FUNCTION_BLOCK Seven_State_Actuator_CAT (* Composite Function Block Type *)
  (* Standard: 61499-2 *)
  (* Version 0.0, 10/7/2025, Schneider Electric, template *)
  PACKAGE Main;
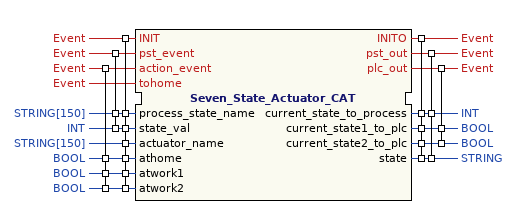
  EVENT_INPUT
    INIT WITH process_state_name, state_val, actuator_name, athome, atwork1, atwork2; (* Initialization Request *)
    pst_event WITH process_state_name, state_val;
    action_event WITH athome, atwork1, atwork2;
    tohome;
  END_EVENT
  EVENT_OUTPUT
    INITO WITH current_state_to_process, current_state1_to_plc, current_state2_to_plc, state; (* Initialization Confirm *)
    pst_out WITH current_state_to_process, state; (* Initialization Confirm *)
    plc_out WITH current_state1_to_plc, current_state2_to_plc;
  END_EVENT
  VAR_INPUT
    process_state_name : STRING[150];
    state_val : INT;
    actuator_name : STRING[150];
    athome : BOOL;
    atwork1 : BOOL;
    atwork2 : BOOL;
  END_VAR
  VAR_OUTPUT
    current_state_to_process : INT; (* Output event qualifier *)
    current_state1_to_plc : BOOL;
    current_state2_to_plc : BOOL;
    state : STRING;
  END_VAR
  FBS
    FB3 : E_DELAY;
    FB4 : SevenStateActuator2;
    FB2 : SELECT_82A43F44E4738F21(IN1 := T#750ms, IN2 := T#500ms); {SET_ATTRIBUTE(Configuration.GenericFBType.InterfaceParams, Runtime.Standard#CNT:=2;SELECT:USINT;IN${CNT$}:TIME)}
    FB5 : ANY2ANY_251AD082F33B40AA3; {SET_ATTRIBUTE(Configuration.GenericFBType.InterfaceParams, Runtime.Standard#CNT:=1;IN${CNT$}:INT;OUT${CNT$}:USINT)}
    IThis : Seven_State_Actuator_CAT_HMI(QI := TRUE);
  END_FBS
  EVENT_CONNECTIONS
    action_event TO FB4.action_event;
    pst_event TO FB4.pst_event;
    FB4.plc_out TO plc_out;
    FB4.pst_out TO pst_out;
    FB4.timer_start TO FB3.START;
    FB3.EO TO FB4.timer_end;
    FB4.timer_stop TO FB3.STOP;
    tohome TO FB4.tohome;
    FB5.CNF TO FB2.REQ;
    FB4.pst_out TO FB5.REQ;
    INIT TO FB4.INIT;
    FB4.INITO TO IThis.INIT;
    FB4.pst_out TO IThis.pst_out;
    FB4.plc_out TO IThis.plc_out;
    IThis.INITO TO INITO;
  END_CONNECTIONS
  DATA_CONNECTIONS
    actuator_name TO FB4.actuator_name;
    state_val TO FB4.state_val;
    process_state_name TO FB4.process_state_name;
    atwork1 TO FB4.atwork1;
    athome TO FB4.athome;
    FB4.current_state_to_pocess TO current_state_to_process;
    FB4.current_state1_to_plc TO current_state1_to_plc;
    FB4.current_state2_to_plc TO current_state2_to_plc;
    atwork2 TO FB4.atwork2;
    FB4.current_state_to_pocess TO FB5.IN1;
    FB5.OUT1 TO FB2.SELECT;
    FB2.OUT TO FB3.DT;
    FB4.state TO state;
    FB4.current_state_to_pocess TO IThis.current_state_to_pocess;
    FB4.current_state1_to_plc TO IThis.current_state1_to_plc;
    FB4.current_state2_to_plc TO IThis.current_state2_to_plc;
  END_CONNECTIONS
END_FUNCTION_BLOCK
